// TwinCAT 3 PLC project Sample01
// ProgramVersion: 3.1.4022.7
// libraries:
//   Tc2_Standard, * (Beckhoff Automation GmbH)
//   Tc2_System, * (Beckhoff Automation GmbH)
//   Tc3_Module, * (Beckhoff Automation GmbH)
// project tree:
//   DUTs/ E_Parity.TcDUT
//   / PlcTask.TcTTO
//   POUs/ FB_SerialCommunication.TcPOU, FB_SerialCommunicationCluster.TcPOU, FB_SerialCommunicationRS232.TcPOU, MAIN.TcPOU
// real-time tasks:
//   TASK PlcTask: cycle T#10ms, priority 20, ADS port 350

CONFIGURATION Sample01
    RESOURCE PLC ON TwinCAT3
        TASK PlcTask(INTERVAL := T#10ms, PRIORITY := 20);
        PROGRAM MAIN WITH PlcTask : MAIN;
    END_RESOURCE
END_CONFIGURATION

// ---- DUTs/E_Parity.TcDUT
{attribute 'qualified_only'}
{attribute 'strict'}
TYPE E_Parity :
(
	None	:= 0,
	Even	:= 1,
	Odd		:= 2,
	Unknown	:= 255
) BYTE := None;
END_TYPE

// ---- POUs/MAIN.TcPOU
PROGRAM MAIN
VAR
	fbSerialCommunication 			: FB_SerialCommunication(nDatabits := 8, eParity := E_Parity.Even, nStopbits := 1);
	fbSerialCommunicationRS232 		: FB_SerialCommunicationRS232(nDatabits := 8, eParity := E_Parity.Even, nStopbits := 1, nBoudRate := 19200);	
	fbSerialCommunicationCluster	: FB_SerialCommunicationCluster(nDatabits := 8, eParity := E_Parity.None, nStopbits := 1);
END_VAR

fbSerialCommunication();
fbSerialCommunicationRS232();
fbSerialCommunicationCluster();

END_PROGRAM

// ---- POUs/FB_SerialCommunication.TcPOU
FUNCTION_BLOCK PUBLIC FB_SerialCommunication
VAR
	nInternalDatabits      : BYTE(7..8);
	eInternalParity        : E_Parity;
	nInternalStopbits	   : BYTE(1..2);	
END_VAR

;

{attribute 'monitoring' := 'call'}
PROPERTY PUBLIC Databits : BYTE(7..8)
GET
Databits := this^.nInternalDatabits;
END_GET
SET
this^.nInternalDatabits := Databits;
END_SET
END_PROPERTY

METHOD FB_init : BOOL
VAR_INPUT
	bInitRetains	: BOOL; // if TRUE, the retain variables are initialized (warm start / cold start)
	bInCopyCode		: BOOL; // if TRUE, the instance afterwards gets moved into the copy code (online change)
	nDatabits    	: BYTE(7..8);
	eParity         : E_Parity;
	nStopbits		: BYTE(1..2);
END_VAR
THIS^.nInternalDatabits := nDatabits;
THIS^.eInternalParity := eParity;
THIS^.nInternalStopbits := nStopbits;
END_METHOD

{attribute 'monitoring' := 'call'}
PROPERTY PUBLIC Parity : E_Parity
GET
Parity := THIS^.eInternalParity;
END_GET
SET
THIS^.eInternalParity := Parity;
END_SET
END_PROPERTY

{attribute 'monitoring' := 'call'}
PROPERTY PUBLIC Stopbits : BYTE(1..2)
GET
Stopbits := THIS^.nInternalStopbits;
END_GET
SET
THIS^.nInternalStopbits := Stopbits;
END_SET
END_PROPERTY

END_FUNCTION_BLOCK

// ---- POUs/FB_SerialCommunicationRS232.TcPOU
FUNCTION_BLOCK PUBLIC FB_SerialCommunicationRS232 EXTENDS FB_SerialCommunication
VAR_INPUT
END_VAR
VAR_OUTPUT
END_VAR
VAR
	nInternalBoudrate	:	UDINT;
END_VAR

METHOD FB_init : BOOL
VAR_INPUT
	bInitRetains	: BOOL; // if TRUE, the retain variables are initialized (warm start / cold start)
	bInCopyCode		: BOOL; // if TRUE, the instance afterwards gets moved into the copy code (online change)
	nDatabits    	: BYTE(7..8);
	eParity         : E_Parity;
	nStopbits		: BYTE(1..2);
	nBoudrate		: UDINT;	
END_VAR
THIS^.nInternalBoudrate := nBoudrate;
END_METHOD

END_FUNCTION_BLOCK

// ---- POUs/FB_SerialCommunicationCluster.TcPOU
FUNCTION_BLOCK PUBLIC FB_SerialCommunicationCluster
VAR	
	fbSerialCommunication01		: FB_SerialCommunication(nDatabits := nInternalDatabits, eParity := eInternalParity, nStopbits := nInternalStopbits);
	fbSerialCommunication02		: FB_SerialCommunication(nDatabits := nInternalDatabits, eParity := eInternalParity, nStopbits := nInternalStopbits);
	nInternalDatabits    		: BYTE(7..8);
	eInternalParity         	: E_Parity;
	nInternalStopbits			: BYTE(1..2);
END_VAR

fbSerialCommunication01();
fbSerialCommunication02();

METHOD FB_init : BOOL
VAR_INPUT
	bInitRetains	: BOOL; // if TRUE, the retain variables are initialized (warm start / cold start)
	bInCopyCode		: BOOL; // if TRUE, the instance afterwards gets moved into the copy code (online change)
	nDatabits    	: BYTE(7..8);
	eParity         : E_Parity;
	nStopbits		: BYTE(1..2);	
END_VAR
fbSerialCommunication01.FB_init(bInitRetains := bInitRetains, bInCopyCode := bInCopyCode, nDatabits := nDatabits, eParity := eParity, nStopbits := nStopbits);
fbSerialCommunication02.FB_init(bInitRetains := bInitRetains, bInCopyCode := bInCopyCode, nDatabits := nDatabits, eParity := eParity, nStopbits := nStopbits);

THIS^.nInternalDatabits := nDatabits;
THIS^.eInternalParity := eParity;
THIS^.nInternalStopbits := nStopbits;
END_METHOD

END_FUNCTION_BLOCK
